FUNCTION_BLOCK FB_CheckFeedback
VAR_INPUT
	t : E_FT;
	bRising: BOOL := TRUE;
END_VAR
VAR_IN_OUT
	FeedbackTimer : TON;
END_VAR
VAR_OUTPUT
	o_nResult : INT := 0;	// -1: fail, 0: checking, 1: success 
END_VAR
VAR
	bFeedback : BOOL;
	nCheckingTime: INT;
	sAlarmMessage: STRING;
	sMsg: INT;
END_VAR

CASE t OF
	E_FT.PUMP:
		bFeedback := GVL_IO.DI_M1;
		
	E_FT.CYL1_E:
		bFeedback := GVL_IO.DI_CYL1_E;
	E_FT.CYL1_R:
		bFeedback := GVL_IO.DI_CYL1_R;
	E_FT.CYL2_E:
		bFeedback := GVL_IO.DI_CYL2_E;
	E_FT.CYL2_R:
		bFeedback := GVL_IO.DI_CYL2_R;
	E_FT.CYL3_E:
		bFeedback := GVL_IO.DI_CYL3_E;
	E_FT.CYL3_R:
		bFeedback := GVL_IO.DI_CYL3_R;
	E_FT.CYL4_E:
		bFeedback := GVL_IO.DI_CYL4_E;
	E_FT.CYL4_R:
		bFeedback := GVL_IO.DI_CYL4_R;
	E_FT.CYL5_E:
		bFeedback := GVL_IO.DI_CYL5_E;
	E_FT.CYL5_R:
		bFeedback := GVL_IO.DI_CYL5_R;
	E_FT.CYL6_E:
		bFeedback := GVL_IO.DI_CYL6_E;
	E_FT.CYL6_R:
		bFeedback := GVL_IO.DI_CYL6_R;
	E_FT.CYL7_E:
		bFeedback := GVL_IO.DI_CYL7_E;
	E_FT.CYL7_R:
		bFeedback := GVL_IO.DI_CYL7_R;
		
	E_FT.PCYL1_E:
		bFeedback := GVL_IO.DI_PCYL1_E;
	E_FT.PCYL1_R:
		bFeedback := GVL_IO.DI_PCYL1_R;
	E_FT.PCYL2_E:
		bFeedback := GVL_IO.DI_PCYL2_E;
	E_FT.PCYL2_R:
		bFeedback := GVL_IO.DI_PCYL2_R;
END_CASE
IF t = E_FT.PUMP THEN
	nCheckingTime := GVL_HMI.i_nPumpFeedbackCheckingTime;
ELSE
	nCheckingTime := GVL_HMI.i_nCylinderFeedbackCheckingTime;
END_IF

IF NOT bRising THEN bFeedback := NOT bFeedback; END_IF

IF NOT bFeedback AND NOT FeedbackTimer.IN THEN
    FeedbackTimer(IN := TRUE, PT := INT_TO_TIME(nCheckingTime));	// T#3S
ELSE
	IF bFeedback THEN
		FeedbackTimer(IN := FALSE);
		o_nResult := 1;
    ELSIF FeedbackTimer.Q THEN
		CASE t OF
			E_FT.PUMP:
				GVL_HMI.i_nPumpState := -1;
				sAlarmMessage := GVL_AlarmMessage.PUMP;
				IF bRising THEN sAlarmMessage := GVL_AlarmMessage.PUMP; ELSE sAlarmMessage := GVL_AlarmMessage.PUMP_OFF; END_IF
				
			E_FT.CYL1_E:
				GVL_HMI.i_nPCylinder1State := -1;
				IF bRising THEN sAlarmMessage := GVL_AlarmMessage.CYL1_NOT_EXTENDED; ELSE sAlarmMessage := GVL_AlarmMessage.CYL1_NOT_EXTENDED_OFF; END_IF
			E_FT.CYL1_R:
				GVL_HMI.i_nCylinder1State := -1;
				IF bRising THEN sAlarmMessage := GVL_AlarmMessage.CYL1_NOT_RETRACTED; ELSE sAlarmMessage := GVL_AlarmMessage.CYL1_NOT_RETRACTED_OFF; END_IF
			E_FT.CYL2_E:
				GVL_HMI.i_nCylinder2State := -1;
				IF bRising THEN sAlarmMessage := GVL_AlarmMessage.CYL2_NOT_EXTENDED; ELSE sAlarmMessage := GVL_AlarmMessage.CYL2_NOT_EXTENDED_OFF; END_IF
			E_FT.CYL2_R:
				GVL_HMI.i_nCylinder2State := -1;
				IF bRising THEN sAlarmMessage := GVL_AlarmMessage.CYL2_NOT_RETRACTED; ELSE sAlarmMessage := GVL_AlarmMessage.CYL2_NOT_RETRACTED_OFF; END_IF
			E_FT.CYL3_E:
				GVL_HMI.i_nCylinder3State := -1;
				IF bRising THEN sAlarmMessage := GVL_AlarmMessage.CYL3_NOT_EXTENDED; ELSE sAlarmMessage := GVL_AlarmMessage.CYL3_NOT_EXTENDED_OFF; END_IF
			E_FT.CYL3_R:
				GVL_HMI.i_nCylinder3State := -1;
				IF bRising THEN sAlarmMessage := GVL_AlarmMessage.CYL3_NOT_RETRACTED; ELSE sAlarmMessage := GVL_AlarmMessage.CYL3_NOT_RETRACTED_OFF; END_IF
			E_FT.CYL4_E:
				GVL_HMI.i_nCylinder4State := -1;
				IF bRising THEN sAlarmMessage := GVL_AlarmMessage.CYL4_NOT_EXTENDED; ELSE sAlarmMessage := GVL_AlarmMessage.CYL4_NOT_EXTENDED_OFF; END_IF
			E_FT.CYL4_R:
				GVL_HMI.i_nCylinder4State := -1;
				IF bRising THEN sAlarmMessage := GVL_AlarmMessage.CYL4_NOT_RETRACTED; ELSE sAlarmMessage := GVL_AlarmMessage.CYL4_NOT_RETRACTED_OFF; END_IF
			E_FT.CYL5_E:
				GVL_HMI.i_nCylinder5State := -1;
				IF bRising THEN sAlarmMessage := GVL_AlarmMessage.CYL5_NOT_EXTENDED; ELSE sAlarmMessage := GVL_AlarmMessage.CYL5_NOT_EXTENDED_OFF; END_IF
			E_FT.CYL5_R:
				GVL_HMI.i_nCylinder5State := -1;
				IF bRising THEN sAlarmMessage := GVL_AlarmMessage.CYL5_NOT_RETRACTED; ELSE sAlarmMessage := GVL_AlarmMessage.CYL5_NOT_RETRACTED_OFF; END_IF
			E_FT.CYL6_E:
				GVL_HMI.i_nCylinder6State := -1;
				IF bRising THEN sAlarmMessage := GVL_AlarmMessage.CYL6_NOT_EXTENDED; ELSE sAlarmMessage := GVL_AlarmMessage.CYL6_NOT_EXTENDED_OFF; END_IF
			E_FT.CYL6_R:
				GVL_HMI.i_nCylinder6State := -1;
				IF bRising THEN sAlarmMessage := GVL_AlarmMessage.CYL6_NOT_RETRACTED; ELSE sAlarmMessage := GVL_AlarmMessage.CYL6_NOT_RETRACTED_OFF; END_IF
			E_FT.CYL7_E:
				GVL_HMI.i_nCylinder7State := -1;
				IF bRising THEN sAlarmMessage := GVL_AlarmMessage.CYL7_NOT_EXTENDED; ELSE sAlarmMessage := GVL_AlarmMessage.CYL7_NOT_EXTENDED_OFF; END_IF
			E_FT.CYL7_R:
				GVL_HMI.i_nCylinder7State := -1;
				IF bRising THEN sAlarmMessage := GVL_AlarmMessage.CYL7_NOT_RETRACTED; ELSE sAlarmMessage := GVL_AlarmMessage.CYL7_NOT_RETRACTED_OFF; END_IF
				
			E_FT.PCYL1_E:
				GVL_HMI.i_nPCylinder1State := -1;
				IF bRising THEN sAlarmMessage := GVL_AlarmMessage.PCYL1_NOT_EXTENDED; ELSE sAlarmMessage := GVL_AlarmMessage.PCYL1_NOT_EXTENDED_OFF; END_IF
			E_FT.PCYL1_R:
				GVL_HMI.i_nPCylinder1State := -1;
				IF bRising THEN sAlarmMessage := GVL_AlarmMessage.PCYL1_NOT_RETRACTED; ELSE sAlarmMessage := GVL_AlarmMessage.PCYL1_NOT_RETRACTED_OFF; END_IF
			E_FT.PCYL2_E:
				GVL_HMI.i_nPCylinder2State := -1;
				IF bRising THEN sAlarmMessage := GVL_AlarmMessage.PCYL2_NOT_EXTENDED; ELSE sAlarmMessage := GVL_AlarmMessage.PCYL2_NOT_EXTENDED_OFF; END_IF
			E_FT.PCYL2_R:
				GVL_HMI.i_nPCylinder2State := -1;
				IF bRising THEN sAlarmMessage := GVL_AlarmMessage.PCYL2_NOT_RETRACTED; ELSE sAlarmMessage := GVL_AlarmMessage.PCYL2_NOT_RETRACTED_OFF; END_IF
		END_CASE
		
		FB_SetAlarm( sMsg := sAlarmMessage );
		o_nResult := -1;
    END_IF
END_IF

END_FUNCTION_BLOCK

(* stored: Version 1.1.0.1, ProductVersion 3.1.4024.6
   POU FB_CheckFeedback: Id {6366c31c-5a01-44e5-9972-875c3b27c878}, SpecialFunc None *)
